(* PLC project Adressering.ecp, WAGO e!COCKPIT e!COCKPIT *)
(* stored: creationDateTime 2021-01-18T14:20:23.2110188, modificationDateTime 2021-01-18T11:51:27.6823754 *)

{attribute 'qualified_only'}
VAR_GLOBAL  (* STLV80_563 *)
  STLV80_A_563_5A201 : dtRomtype_0;  (* Gang *)
  STLV80_A_563_5A202 : dtRomtype_1;  (* kontor *)
  STLV80_A_563_5A203 : dtRomtype_2;  (* Teamkontor *)
  STLV80_A_563_5A204 : dtRomtype_3;  (* FellesRom *)
  STLV80_A_563_5B201 : dtRomtype_4;  (* BEV *)
  STLV80_A_563_5C301 : dtRomtype_5;  (* BEV *)
  STLV80_A_563_5D301 : dtRomtype_6;  (* TEST *)
  STLV80_A_563_5E201 : dtRomtype_7;  (* test *)
  STLV80_A_563_5E301 : dtRomtype_8;  (* TEST *)
  STLV80_A_563_5F201 : dtRomtype_9;  (* TEST *)
  STLV80_A_563_5F202 : dtRomtype_10;  (* TEST *)
  STLV80_A_563_5F203 : dtRomtype_11;  (* TEST *)
  STLV80_A_563_5F204 : dtRomtype_12;  (* TEST *)
END_VAR

PROGRAM PRG_563_KNX
  VAR
    i : INT := 0;  (* Felles *)
    Interval : OSCAT_BASIC.CLK_PRG;
    typDPT : typDPT;
    M1_001_5A201_RB601_V : fbDPT_Switch_pro;
    M1_002_5A201_RB601_HVAC : fbDPT_Switch_pro;
    M1_003_5A202_RT601_CT : fbDPT_Value_Temp_pro;  (* 5A202 *)
    M1_004_5A202_RB601_V : fbDPT_Switch_pro;
    M1_005_5A202_RB601_HVAC : fbDPT_Switch_pro;
    M1_006_5A203_RT601_CT : fbDPT_Value_Temp_pro;  (* 5A203 *)
    M1_007_5A203_RB601_V : fbDPT_Switch_pro;
    M1_008_5A203_LH601_OP : fbDPT_Scaling_pro;
    M1_009_5A203_RB601_HVAC : fbDPT_Switch_pro;
    M1_010_5A204_RT601_CT : fbDPT_Value_Temp_pro;  (* 5A204 *)
    M1_011_5A204_RB601_V : fbDPT_Switch_pro;
    M1_012_5A204_RB601_HVAC : fbDPT_Switch_pro;
    M1_013_5A204_LC601_OP : fbDPT_Scaling_pro;
    M1_014_5B201_RT601_CT : fbDPT_Value_Temp_pro;  (* 5B201 *)
    M1_015_5B201_RB601_V : fbDPT_Switch_pro;
    M1_016_5B201_RB601_HVAC : fbDPT_Switch_pro;
    M1_017_5B201_RY601_CV : fbDPT_Value_AirQuality_pro;
    M1_018_5C301_RT601_CT : fbDPT_Value_Temp_pro;  (* 5C301 *)
    M1_019_5C301_RB601_V : fbDPT_Switch_pro;
    M1_020_5C301_LH601_OP : fbDPT_Scaling_pro;
    M1_021_5C301_RB601_HVAC : fbDPT_Switch_pro;
    M1_022_5C301_LC601_OP : fbDPT_Scaling_pro;
    M1_023_5D301_RT601_CT : fbDPT_Value_Temp_pro;  (* 5D301 *)
    M1_024_5D301_RB601_V : fbDPT_Switch_pro;
    M1_025_5D301_LH601_OP : fbDPT_Scaling_pro;
    M1_026_5D301_RB601_HVAC : fbDPT_Switch_pro;
    M1_027_5D301_RY601_CV : fbDPT_Value_AirQuality_pro;
    M1_028_5E201_RT601_CT : fbDPT_Value_Temp_pro;  (* 5E201 *)
    M1_029_5E201_RB601_V : fbDPT_Switch_pro;
    M1_030_5E201_RB601_HVAC : fbDPT_Switch_pro;
    M1_031_5E201_LC601_OP : fbDPT_Scaling_pro;
    M1_032_5E201_RY601_CV : fbDPT_Value_AirQuality_pro;
    M1_033_5E301_RT601_CT : fbDPT_Value_Temp_pro;  (* 5E301 *)
    M1_034_5E301_RB601_V : fbDPT_Switch_pro;
    M1_035_5E301_LH601_OP : fbDPT_Scaling_pro;
    M1_036_5E301_RB601_HVAC : fbDPT_Switch_pro;
    M1_037_5E301_LC601_OP : fbDPT_Scaling_pro;
    M1_038_5E301_RY601_CV : fbDPT_Value_AirQuality_pro;
    M1_039_5F201_RT601_CT : fbDPT_Value_Temp_pro;  (* 5F201 *)
    M1_040_5F201_RB601_V : fbDPT_Switch_pro;
    M1_041_5F201_LH601_OP : fbDPT_Scaling_pro;
    M1_042_5F201_RB601_HVAC : fbDPT_Switch_pro;
    M1_043_5F201_RT601_SP_FB : fbDPT_Value_Temp_pro;
    M1_044_5F201_RT601_SP : fbDPT_Value_Temp_pro;
    M1_045_5F202_RT601_CT : fbDPT_Value_Temp_pro;  (* 5F202 *)
    M1_046_5F202_RB601_V : fbDPT_Switch_pro;
    M1_047_5F202_LH601_OP : fbDPT_Scaling_pro;
    M1_048_5F202_RB601_HVAC : fbDPT_Switch_pro;
    M1_049_5F202_LC601_OP : fbDPT_Scaling_pro;
    M1_050_5F202_RT601_SP_FB : fbDPT_Value_Temp_pro;
    M1_051_5F202_RT601_SP : fbDPT_Value_Temp_pro;
    M1_052_5F203_RT601_CT : fbDPT_Value_Temp_pro;  (* 5F203 *)
    M1_053_5F203_RB601_V : fbDPT_Switch_pro;
    M1_054_5F203_LH601_OP : fbDPT_Scaling_pro;
    M1_055_5F203_RB601_HVAC : fbDPT_Switch_pro;
    M1_056_5F203_RY601_CV : fbDPT_Value_AirQuality_pro;
    M1_057_5F203_RT601_SP_FB : fbDPT_Value_Temp_pro;
    M1_058_5F203_RT601_SP : fbDPT_Value_Temp_pro;
    M1_059_5F204_RT601_CT : fbDPT_Value_Temp_pro;  (* 5F204 *)
    M1_060_5F204_RB601_V : fbDPT_Switch_pro;
    M1_061_5F204_LH601_OP : fbDPT_Scaling_pro;
    M1_062_5F204_RB601_HVAC : fbDPT_Switch_pro;
    M1_063_5F204_LC601_OP : fbDPT_Scaling_pro;
    M1_064_5F204_RY601_CV : fbDPT_Value_AirQuality_pro;
    M1_065_5F204_RT601_SP_FB : fbDPT_Value_Temp_pro;
    M1_066_5F204_RT601_SP : fbDPT_Value_Temp_pro;
  END_VAR
  VAR  (* added by the conversion: wires and edge detectors of the diagram *)
    _ADD9_OUT : INT;
    _GT15_OUT : BOOL;
    _MOVE19_ENO : BOOL;
    _MOVE19_OUT : INT;
  END_VAR

(* CFC diagram, written out as Structured Text *)
(* KNX Sending interval *)
Interval(PT := t#2M);
_ADD9_OUT := BOOL_TO_INT(Interval.Q) + i;
i := _ADD9_OUT;
_GT15_OUT := i > 14;
_MOVE19_OUT := MOVE(EN := _GT15_OUT, IN := 0, ENO => _MOVE19_ENO);
IF _MOVE19_ENO THEN i := _MOVE19_OUT; END_IF;
(* Rom 5A201 *)
(* RB601_V *)
M1_001_5A201_RB601_V(bPortKNX := 1, dwIndex_DPT := 1, typDPT := typDPT);
STLV80_563.STLV80_A_563_5A201.RB601_V := M1_001_5A201_RB601_V.xSwitch_OUT;
(* RB601_HVAC *)
M1_002_5A201_RB601_HVAC(bPortKNX := 1, dwIndex_DPT := 2, typDPT := typDPT);
STLV80_563.STLV80_A_563_5A201.RB601_HVAC := M1_002_5A201_RB601_HVAC.xSwitch_OUT;
(* Rom 5A202 *)
(* RT601_CT *)
(* RB601_V *)
M1_003_5A202_RT601_CT(bPortKNX := 1, dwIndex_DPT := 3, typDPT := typDPT);
STLV80_563.STLV80_A_563_5A202.RT601_CT := M1_003_5A202_RT601_CT.rValue_OUT;
M1_004_5A202_RB601_V(bPortKNX := 1, dwIndex_DPT := 4, typDPT := typDPT);
STLV80_563.STLV80_A_563_5A202.RB601_V := M1_004_5A202_RB601_V.xSwitch_OUT;
(* RB601_HVAC *)
M1_005_5A202_RB601_HVAC(bPortKNX := 1, dwIndex_DPT := 5, typDPT := typDPT);
STLV80_563.STLV80_A_563_5A202.RB601_HVAC := M1_005_5A202_RB601_HVAC.xSwitch_OUT;
(* Rom 5A203 *)
(* RT601_CT *)
(* RB601_V *)
M1_006_5A203_RT601_CT(bPortKNX := 1, dwIndex_DPT := 6, typDPT := typDPT);
STLV80_563.STLV80_A_563_5A203.RT601_CT := M1_006_5A203_RT601_CT.rValue_OUT;
M1_007_5A203_RB601_V(bPortKNX := 1, dwIndex_DPT := 7, typDPT := typDPT);
STLV80_563.STLV80_A_563_5A203.RB601_V := M1_007_5A203_RB601_V.xSwitch_OUT;
(* LH601_OP *)
(* RB601_HVAC *)
M1_008_5A203_LH601_OP(bPortKNX := 1, dwIndex_DPT := 8, rValue_IN := STLV80_563.STLV80_A_563_5A203.LH601_OP, xUpdate_KNX := i = 0, typDPT := typDPT);
M1_009_5A203_RB601_HVAC(bPortKNX := 1, dwIndex_DPT := 9, typDPT := typDPT);
STLV80_563.STLV80_A_563_5A203.RB601_HVAC := M1_009_5A203_RB601_HVAC.xSwitch_OUT;
(* Rom 5A204 *)
(* RT601_CT *)
(* RB601_V *)
M1_010_5A204_RT601_CT(bPortKNX := 1, dwIndex_DPT := 10, typDPT := typDPT);
STLV80_563.STLV80_A_563_5A204.RT601_CT := M1_010_5A204_RT601_CT.rValue_OUT;
M1_011_5A204_RB601_V(bPortKNX := 1, dwIndex_DPT := 11, typDPT := typDPT);
STLV80_563.STLV80_A_563_5A204.RB601_V := M1_011_5A204_RB601_V.xSwitch_OUT;
(* RB601_HVAC *)
M1_012_5A204_RB601_HVAC(bPortKNX := 1, dwIndex_DPT := 12, typDPT := typDPT);
STLV80_563.STLV80_A_563_5A204.RB601_HVAC := M1_012_5A204_RB601_HVAC.xSwitch_OUT;
(* LC601_OP *)
M1_013_5A204_LC601_OP(bPortKNX := 1, dwIndex_DPT := 13, rValue_IN := STLV80_563.STLV80_A_563_5A204.LC601_OP, xUpdate_KNX := i = 1, typDPT := typDPT);
(* Rom 5B201 *)
(* RT601_CT *)
(* RB601_V *)
M1_014_5B201_RT601_CT(bPortKNX := 1, dwIndex_DPT := 14, typDPT := typDPT);
STLV80_563.STLV80_A_563_5B201.RT601_CT := M1_014_5B201_RT601_CT.rValue_OUT;
M1_015_5B201_RB601_V(bPortKNX := 1, dwIndex_DPT := 15, typDPT := typDPT);
STLV80_563.STLV80_A_563_5B201.RB601_V := M1_015_5B201_RB601_V.xSwitch_OUT;
(* RB601_HVAC *)
M1_016_5B201_RB601_HVAC(bPortKNX := 1, dwIndex_DPT := 16, typDPT := typDPT);
STLV80_563.STLV80_A_563_5B201.RB601_HVAC := M1_016_5B201_RB601_HVAC.xSwitch_OUT;
(* RY601_CV *)
M1_017_5B201_RY601_CV(bPortKNX := 1, dwIndex_DPT := 17, typDPT := typDPT);
STLV80_563.STLV80_A_563_5B201.RY601_CV := M1_017_5B201_RY601_CV.rValue_OUT;
(* Rom 5C301 *)
(* RT601_CT *)
(* RB601_V *)
M1_018_5C301_RT601_CT(bPortKNX := 1, dwIndex_DPT := 18, typDPT := typDPT);
STLV80_563.STLV80_A_563_5C301.RT601_CT := M1_018_5C301_RT601_CT.rValue_OUT;
M1_019_5C301_RB601_V(bPortKNX := 1, dwIndex_DPT := 19, typDPT := typDPT);
STLV80_563.STLV80_A_563_5C301.RB601_V := M1_019_5C301_RB601_V.xSwitch_OUT;
(* LH601_OP *)
(* RB601_HVAC *)
M1_020_5C301_LH601_OP(bPortKNX := 1, dwIndex_DPT := 20, rValue_IN := STLV80_563.STLV80_A_563_5C301.LH601_OP, xUpdate_KNX := i = 2, typDPT := typDPT);
M1_021_5C301_RB601_HVAC(bPortKNX := 1, dwIndex_DPT := 21, typDPT := typDPT);
STLV80_563.STLV80_A_563_5C301.RB601_HVAC := M1_021_5C301_RB601_HVAC.xSwitch_OUT;
(* LC601_OP *)
M1_022_5C301_LC601_OP(bPortKNX := 1, dwIndex_DPT := 22, rValue_IN := STLV80_563.STLV80_A_563_5C301.LC601_OP, xUpdate_KNX := i = 3, typDPT := typDPT);
(* Rom 5D301 *)
(* RT601_CT *)
(* RB601_V *)
M1_023_5D301_RT601_CT(bPortKNX := 1, dwIndex_DPT := 23, typDPT := typDPT);
STLV80_563.STLV80_A_563_5D301.RT601_CT := M1_023_5D301_RT601_CT.rValue_OUT;
M1_024_5D301_RB601_V(bPortKNX := 1, dwIndex_DPT := 24, typDPT := typDPT);
STLV80_563.STLV80_A_563_5D301.RB601_V := M1_024_5D301_RB601_V.xSwitch_OUT;
(* LH601_OP *)
(* RB601_HVAC *)
M1_025_5D301_LH601_OP(bPortKNX := 1, dwIndex_DPT := 25, rValue_IN := STLV80_563.STLV80_A_563_5D301.LH601_OP, xUpdate_KNX := i = 4, typDPT := typDPT);
M1_026_5D301_RB601_HVAC(bPortKNX := 1, dwIndex_DPT := 26, typDPT := typDPT);
STLV80_563.STLV80_A_563_5D301.RB601_HVAC := M1_026_5D301_RB601_HVAC.xSwitch_OUT;
(* RY601_CV *)
M1_027_5D301_RY601_CV(bPortKNX := 1, dwIndex_DPT := 27, typDPT := typDPT);
STLV80_563.STLV80_A_563_5D301.RY601_CV := M1_027_5D301_RY601_CV.rValue_OUT;
(* Rom 5E201 *)
(* RT601_CT *)
(* RB601_V *)
M1_028_5E201_RT601_CT(bPortKNX := 1, dwIndex_DPT := 28, typDPT := typDPT);
STLV80_563.STLV80_A_563_5E201.RT601_CT := M1_028_5E201_RT601_CT.rValue_OUT;
M1_029_5E201_RB601_V(bPortKNX := 1, dwIndex_DPT := 29, typDPT := typDPT);
STLV80_563.STLV80_A_563_5E201.RB601_V := M1_029_5E201_RB601_V.xSwitch_OUT;
(* RB601_HVAC *)
M1_030_5E201_RB601_HVAC(bPortKNX := 1, dwIndex_DPT := 30, typDPT := typDPT);
STLV80_563.STLV80_A_563_5E201.RB601_HVAC := M1_030_5E201_RB601_HVAC.xSwitch_OUT;
(* LC601_OP *)
(* RY601_CV *)
M1_031_5E201_LC601_OP(bPortKNX := 1, dwIndex_DPT := 31, rValue_IN := STLV80_563.STLV80_A_563_5E201.LC601_OP, xUpdate_KNX := i = 5, typDPT := typDPT);
M1_032_5E201_RY601_CV(bPortKNX := 1, dwIndex_DPT := 32, typDPT := typDPT);
STLV80_563.STLV80_A_563_5E201.RY601_CV := M1_032_5E201_RY601_CV.rValue_OUT;
(* Rom 5E301 *)
(* RT601_CT *)
(* RB601_V *)
M1_033_5E301_RT601_CT(bPortKNX := 1, dwIndex_DPT := 33, typDPT := typDPT);
STLV80_563.STLV80_A_563_5E301.RT601_CT := M1_033_5E301_RT601_CT.rValue_OUT;
M1_034_5E301_RB601_V(bPortKNX := 1, dwIndex_DPT := 34, typDPT := typDPT);
STLV80_563.STLV80_A_563_5E301.RB601_V := M1_034_5E301_RB601_V.xSwitch_OUT;
(* LH601_OP *)
(* RB601_HVAC *)
M1_035_5E301_LH601_OP(bPortKNX := 1, dwIndex_DPT := 35, rValue_IN := STLV80_563.STLV80_A_563_5E301.LH601_OP, xUpdate_KNX := i = 6, typDPT := typDPT);
M1_036_5E301_RB601_HVAC(bPortKNX := 1, dwIndex_DPT := 36, typDPT := typDPT);
STLV80_563.STLV80_A_563_5E301.RB601_HVAC := M1_036_5E301_RB601_HVAC.xSwitch_OUT;
(* LC601_OP *)
(* RY601_CV *)
M1_037_5E301_LC601_OP(bPortKNX := 1, dwIndex_DPT := 37, rValue_IN := STLV80_563.STLV80_A_563_5E301.LC601_OP, xUpdate_KNX := i = 7, typDPT := typDPT);
M1_038_5E301_RY601_CV(bPortKNX := 1, dwIndex_DPT := 38, typDPT := typDPT);
STLV80_563.STLV80_A_563_5E301.RY601_CV := M1_038_5E301_RY601_CV.rValue_OUT;
(* Rom 5F201 *)
(* RT601_CT *)
(* RB601_V *)
M1_039_5F201_RT601_CT(bPortKNX := 1, dwIndex_DPT := 39, typDPT := typDPT);
STLV80_563.STLV80_A_563_5F201.RT601_CT := M1_039_5F201_RT601_CT.rValue_OUT;
M1_040_5F201_RB601_V(bPortKNX := 1, dwIndex_DPT := 40, typDPT := typDPT);
STLV80_563.STLV80_A_563_5F201.RB601_V := M1_040_5F201_RB601_V.xSwitch_OUT;
(* LH601_OP *)
(* RB601_HVAC *)
M1_041_5F201_LH601_OP(bPortKNX := 1, dwIndex_DPT := 41, rValue_IN := STLV80_563.STLV80_A_563_5F201.LH601_OP, xUpdate_KNX := i = 8, typDPT := typDPT);
M1_042_5F201_RB601_HVAC(bPortKNX := 1, dwIndex_DPT := 42, typDPT := typDPT);
STLV80_563.STLV80_A_563_5F201.RB601_HVAC := M1_042_5F201_RB601_HVAC.xSwitch_OUT;
(* RT601_SP Feedback *)
(* RT601_SP *)
M1_043_5F201_RT601_SP_FB(bPortKNX := 1, dwIndex_DPT := 43, typDPT := typDPT);
STLV80_563.STLV80_A_563_5F201.RT601_SP_IN := M1_043_5F201_RT601_SP_FB.rValue_OUT;
M1_044_5F201_RT601_SP(bPortKNX := 1, dwIndex_DPT := 44, rValue_IN := STLV80_563.STLV80_A_563_5F201.RT601_SP_D, xUpdate_KNX := NOT STLV80_563.STLV80_A_563_5F201.RB601_HVAC, typDPT := typDPT);
(* Rom 5F202 *)
(* RT601_CT *)
(* RB601_V *)
M1_045_5F202_RT601_CT(bPortKNX := 1, dwIndex_DPT := 45, typDPT := typDPT);
STLV80_563.STLV80_A_563_5F202.RT601_CT := M1_045_5F202_RT601_CT.rValue_OUT;
M1_046_5F202_RB601_V(bPortKNX := 1, dwIndex_DPT := 46, typDPT := typDPT);
STLV80_563.STLV80_A_563_5F202.RB601_V := M1_046_5F202_RB601_V.xSwitch_OUT;
(* LH601_OP *)
(* RB601_HVAC *)
M1_047_5F202_LH601_OP(bPortKNX := 1, dwIndex_DPT := 47, rValue_IN := STLV80_563.STLV80_A_563_5F202.LH601_OP, xUpdate_KNX := i = 9, typDPT := typDPT);
M1_048_5F202_RB601_HVAC(bPortKNX := 1, dwIndex_DPT := 48, typDPT := typDPT);
STLV80_563.STLV80_A_563_5F202.RB601_HVAC := M1_048_5F202_RB601_HVAC.xSwitch_OUT;
(* LC601_OP *)
M1_049_5F202_LC601_OP(bPortKNX := 1, dwIndex_DPT := 49, rValue_IN := STLV80_563.STLV80_A_563_5F202.LC601_OP, xUpdate_KNX := i = 10, typDPT := typDPT);
(* RT601_SP Feedback *)
(* RT601_SP *)
M1_050_5F202_RT601_SP_FB(bPortKNX := 1, dwIndex_DPT := 50, typDPT := typDPT);
STLV80_563.STLV80_A_563_5F202.RT601_SP_IN := M1_050_5F202_RT601_SP_FB.rValue_OUT;
M1_051_5F202_RT601_SP(bPortKNX := 1, dwIndex_DPT := 51, rValue_IN := STLV80_563.STLV80_A_563_5F202.RT601_SP_D, xUpdate_KNX := NOT STLV80_563.STLV80_A_563_5F202.RB601_HVAC, typDPT := typDPT);
(* Rom 5F203 *)
(* RT601_CT *)
(* RB601_V *)
M1_052_5F203_RT601_CT(bPortKNX := 1, dwIndex_DPT := 52, typDPT := typDPT);
STLV80_563.STLV80_A_563_5F203.RT601_CT := M1_052_5F203_RT601_CT.rValue_OUT;
M1_053_5F203_RB601_V(bPortKNX := 1, dwIndex_DPT := 53, typDPT := typDPT);
STLV80_563.STLV80_A_563_5F203.RB601_V := M1_053_5F203_RB601_V.xSwitch_OUT;
(* LH601_OP *)
(* RB601_HVAC *)
M1_054_5F203_LH601_OP(bPortKNX := 1, dwIndex_DPT := 54, rValue_IN := STLV80_563.STLV80_A_563_5F203.LH601_OP, xUpdate_KNX := i = 11, typDPT := typDPT);
M1_055_5F203_RB601_HVAC(bPortKNX := 1, dwIndex_DPT := 55, typDPT := typDPT);
STLV80_563.STLV80_A_563_5F203.RB601_HVAC := M1_055_5F203_RB601_HVAC.xSwitch_OUT;
(* RY601_CV *)
M1_056_5F203_RY601_CV(bPortKNX := 1, dwIndex_DPT := 56, typDPT := typDPT);
STLV80_563.STLV80_A_563_5F203.RY601_CV := M1_056_5F203_RY601_CV.rValue_OUT;
(* RT601_SP Feedback *)
(* RT601_SP *)
M1_057_5F203_RT601_SP_FB(bPortKNX := 1, dwIndex_DPT := 57, typDPT := typDPT);
STLV80_563.STLV80_A_563_5F203.RT601_SP_IN := M1_057_5F203_RT601_SP_FB.rValue_OUT;
M1_058_5F203_RT601_SP(bPortKNX := 1, dwIndex_DPT := 58, rValue_IN := STLV80_563.STLV80_A_563_5F203.RT601_SP_D, xUpdate_KNX := NOT STLV80_563.STLV80_A_563_5F203.RB601_HVAC, typDPT := typDPT);
(* Rom 5F204 *)
(* RT601_CT *)
(* RB601_V *)
M1_059_5F204_RT601_CT(bPortKNX := 1, dwIndex_DPT := 59, typDPT := typDPT);
STLV80_563.STLV80_A_563_5F204.RT601_CT := M1_059_5F204_RT601_CT.rValue_OUT;
M1_060_5F204_RB601_V(bPortKNX := 1, dwIndex_DPT := 60, typDPT := typDPT);
STLV80_563.STLV80_A_563_5F204.RB601_V := M1_060_5F204_RB601_V.xSwitch_OUT;
(* LH601_OP *)
(* RB601_HVAC *)
M1_061_5F204_LH601_OP(bPortKNX := 1, dwIndex_DPT := 61, rValue_IN := STLV80_563.STLV80_A_563_5F204.LH601_OP, xUpdate_KNX := i = 12, typDPT := typDPT);
M1_062_5F204_RB601_HVAC(bPortKNX := 1, dwIndex_DPT := 62, typDPT := typDPT);
STLV80_563.STLV80_A_563_5F204.RB601_HVAC := M1_062_5F204_RB601_HVAC.xSwitch_OUT;
(* LC601_OP *)
(* RY601_CV *)
M1_063_5F204_LC601_OP(bPortKNX := 1, dwIndex_DPT := 63, rValue_IN := STLV80_563.STLV80_A_563_5F204.LC601_OP, xUpdate_KNX := i = 13, typDPT := typDPT);
M1_064_5F204_RY601_CV(bPortKNX := 1, dwIndex_DPT := 64, typDPT := typDPT);
STLV80_563.STLV80_A_563_5F204.RY601_CV := M1_064_5F204_RY601_CV.rValue_OUT;
(* RT601_SP Feedback *)
(* RT601_SP *)
M1_065_5F204_RT601_SP_FB(bPortKNX := 1, dwIndex_DPT := 65, typDPT := typDPT);
STLV80_563.STLV80_A_563_5F204.RT601_SP_IN := M1_065_5F204_RT601_SP_FB.rValue_OUT;
M1_066_5F204_RT601_SP(bPortKNX := 1, dwIndex_DPT := 66, rValue_IN := STLV80_563.STLV80_A_563_5F204.RT601_SP_D, xUpdate_KNX := NOT STLV80_563.STLV80_A_563_5F204.RB601_HVAC, typDPT := typDPT);
END_PROGRAM
